// TIA Portal project "Asenkron Motor Frekans Ayarlama_V17" (V17)

(* hardware
DEVICE "S7-1200 station_1"  S7-1200 Station
   slot 0: "Rack_0"  S7-1200 Rack  Rack  V1.0
   slot 1: "PLC_1"  CPU 1214C DC/DC/DC  6ES7 214-1AG40-0XB0  V4.2
   slot 2: "AQ 4x14BIT_1"  6ES7 232-4HD32-0XB0  V2.0
*)

// ===== PLC "PLC_1"  CPU 1214C DC/DC/DC =====

VAR_GLOBAL   // PLC tag table "Default tag table"
   "STOP" AT %I0.0 : Bool;
   "START" AT %I0.1 : Bool;
   "YARDIMCI1" AT %M0.0 : Bool;
   "YARDIMCI2" AT %M0.1 : Bool;
   "YARDIMCI3" AT %M0.2 : Bool;
   "Sensör1" AT %I0.2 : Bool;
   "Sensör2" AT %I0.3 : Bool;
   "Start Buton" AT %Q0.0 : Bool;
   "Tag_1" AT %MW10 : Int;
   "ACİL STOP" AT %I0.4 : Bool;
   "Analog Çıkış" AT %QW96 : Int;
   "YARDIMCI 4" AT %M0.3 : Bool;
   "Tag_8" AT %M0.4 : Bool;
   "yardımcı5" AT %M0.5 : Bool;
   "yardımcı6" AT %M0.6 : Bool;
   "yardımcı7" AT %M0.7 : Bool;
END_VAR

// folder: System blocks/Program resources

DATA_BLOCK "Timer"   // DB1
{ S7_Optimized_Access := 'TRUE' }
AUTHOR : Simatic
FAMILY : IEC
NAME : IEC_TMR
VERSION : 1.0
// stored: InstanceOfName IEC_TIMER
"IEC_TIMER"
BEGIN
   PT := T#5s;
END_DATA_BLOCK

// folder: (top level)

ORGANIZATION_BLOCK "Main"   // OB1, LAD, ProgramCycle
TITLE = "Main Program Sweep (Cycle)"
{ S7_Optimized_Access := 'TRUE' }
VERSION : 0.1
   VAR_INPUT
      Initial_Call : Bool;   // Initial call of this OB
      Remanence : Bool;   // =True, if remanent data are available
   END_VAR
   VAR_TEMP   // added for the SCL form of the ladder/FBD networks
      _w1 : Bool;
      _w2 : Bool;
      _w3 : Bool;
      _w4 : Bool;
   END_VAR
BEGIN

REGION Network 1
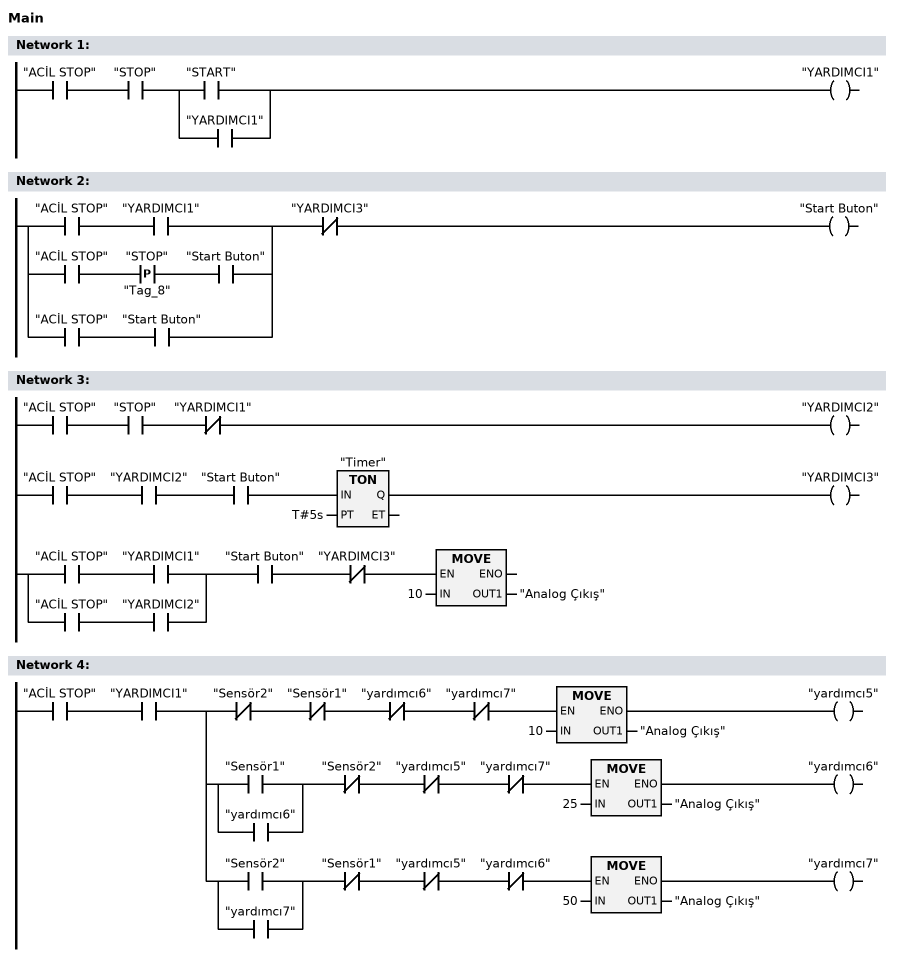
   RUNG wire#powerrail
      Contact( "ACİL STOP" )
      Contact( "STOP" )
      wire#w1
      Contact( "START" )
      wire#w2
      Coil( "YARDIMCI1" )
   END_RUNG
   RUNG wire#w1
      Contact( "YARDIMCI1" )
   END_RUNG wire#w2
   // the same network as SCL:
   "YARDIMCI1" := "ACİL STOP" AND "STOP" AND ("START" OR "YARDIMCI1");
END_REGION

REGION Network 2
   RUNG wire#powerrail
      Contact( "ACİL STOP" )
      Contact( "YARDIMCI1" )
      wire#w1
      I_Contact( "YARDIMCI3" )
      Coil( "Start Buton" )
   END_RUNG
   RUNG wire#powerrail
      Contact( "ACİL STOP" )
      P_Contact(operand := "STOP", bit := "Tag_8")
      Contact( "Start Buton" )
   END_RUNG wire#w1
   RUNG wire#powerrail
      Contact( "ACİL STOP" )
      Contact( "Start Buton" )
   END_RUNG wire#w1
   // the same network as SCL:
   #_w1 := "ACİL STOP" AND "STOP" AND NOT "Tag_8";   // rising edge of "STOP"
   "Tag_8" := "STOP";
   "Start Buton" := (("ACİL STOP" AND "YARDIMCI1") OR (#_w1 AND "Start Buton") OR ("ACİL STOP" AND "Start Buton")) AND NOT "YARDIMCI3";
END_REGION

REGION Network 3
   "YARDIMCI2" := "ACİL STOP" AND "STOP" AND NOT "YARDIMCI1";
   "Timer".TON(IN := "ACİL STOP" AND "YARDIMCI2" AND "Start Buton", PT := T#5s);
   "YARDIMCI3" := "Timer".Q;
   IF (("ACİL STOP" AND "YARDIMCI1") OR ("ACİL STOP" AND "YARDIMCI2")) AND "Start Buton" AND NOT "YARDIMCI3" THEN
       "Analog Çıkış" := 10;
   END_IF;
END_REGION

REGION Network 4
   RUNG wire#powerrail
      Contact( "ACİL STOP" )
      Contact( "YARDIMCI1" )
      wire#w1
      I_Contact( "Sensör2" )
      I_Contact( "Sensör1" )
      I_Contact( "yardımcı6" )
      I_Contact( "yardımcı7" )
      Move(in := 10, out1 => "Analog Çıkış")
      Coil( "yardımcı5" )
   END_RUNG
   RUNG wire#w1
      Contact( "Sensör1" )
      wire#w2
      I_Contact( "Sensör2" )
      I_Contact( "yardımcı5" )
      I_Contact( "yardımcı7" )
      Move(in := 25, out1 => "Analog Çıkış")
      Coil( "yardımcı6" )
   END_RUNG
   RUNG wire#w1
      Contact( "yardımcı6" )
   END_RUNG wire#w2
   RUNG wire#w1
      Contact( "Sensör2" )
      wire#w3
      I_Contact( "Sensör1" )
      I_Contact( "yardımcı5" )
      I_Contact( "yardımcı6" )
      Move(in := 50, out1 => "Analog Çıkış")
      Coil( "yardımcı7" )
   END_RUNG
   RUNG wire#w1
      Contact( "yardımcı7" )
   END_RUNG wire#w3
   // the same network as SCL:
   #_w1 := "ACİL STOP" AND "YARDIMCI1";
   #_w2 := #_w1 AND NOT "Sensör2" AND NOT "Sensör1" AND NOT "yardımcı6" AND NOT "yardımcı7";
   IF #_w2 THEN "Analog Çıkış" := 10; END_IF;
   "yardımcı5" := #_w2;
   #_w3 := #_w1 AND ("Sensör1" OR "yardımcı6") AND NOT "Sensör2" AND NOT "yardımcı5" AND NOT "yardımcı7";
   IF #_w3 THEN "Analog Çıkış" := 25; END_IF;
   "yardımcı6" := #_w3;
   #_w4 := #_w1 AND ("Sensör2" OR "yardımcı7") AND NOT "Sensör1" AND NOT "yardımcı5" AND NOT "yardımcı6";
   IF #_w4 THEN "Analog Çıkış" := 50; END_IF;
   "yardımcı7" := #_w4;
END_REGION
END_ORGANIZATION_BLOCK